INTERFACE I_ParamSaveRestore EXTENDS I_Output

METHOD RestoreAxisParams
VAR_INPUT
END_VAR
END_METHOD

METHOD SaveAxisParams
VAR_INPUT
    Enable : BOOL;
END_VAR
END_METHOD

PROPERTY SavedPosition : LREAL
GET
END_GET
END_PROPERTY

END_INTERFACE

(* stored: Version 1.1.0.1
   Itf I_ParamSaveRestore: Id {f91fa392-42b9-4cf5-a843-28456ed2820b}
   Method RestoreAxisParams: Id {507dd76e-711b-4765-ae75-25397b03046b}
   Method SaveAxisParams: Id {543b2f95-a551-4fd8-9961-1f96cda4fa13}
   Property SavedPosition: Id {3eb2be5e-1bc5-4267-9504-fd4efa432df8}
   Get Get: Id {3d3eebab-1130-4c6e-a759-bbdd38ce8881} *)
